FUNCTION_BLOCK DataManager EXTENDS TcoData.TcoDataExchange
VAR
    _data : stProcessData;
END_VAR

SUPER^();

PROPERTY Data : REFERENCE TO stProcessData
GET
DATA REF= _data;
END_GET
END_PROPERTY

END_FUNCTION_BLOCK

(* stored: Version 1.1.0.1, ProductVersion 3.1.4024.6
   POU DataManager: Id {459b1dbb-712a-0cd3-3b3e-853e1e37477a}, SpecialFunc None
   Property Data: Id {74fa38ed-c762-0ed8-0b5d-76763111150a}
   Get Get: Id {404899c1-174f-00a2-1f16-bae66aacd69f} *)
